Staubli VAL3: oShutter.pgx

public program oShutter(num nChoice (dimensions=1))
// oShutter
begin
  dioSet(oShutter,nChoice)
end
